bacnetModbusDamperInterop[1][22](
  AI_Volume					:= A_360_01_SQ5_C411_VOL,
  AV_CurrentSetpoint			:= A_360_01_SQ5_C411_SP,
  AV_vMin					:= A_360_01_SQ5_C411_VMIN,
  AV_vMax					:= A_360_01_SQ5_C411_VMAX,
  AI_Position				:= A_360_01_SQ5_C411_FB,
  AV_ControlledVariable		:= A_360_01_SQ5_C411_C,
  AV_ManualOverride			:= A_360_01_SQ5_C411_KMD,
  BV_ExcludeFromOptimizer	:= A_360_01_SQ5_C411_OPT_EKSKL,
  BV_DamperError				:= A_360_01_SQ5_C411_A1,
  BV_CommunicationError		:= A_360_01_SQ5_C411_A2,
  modbusHoldingRegisters		:= ADR(GVL_Modbus.awHoldingRegisters[i * 30]), 
  modbusCoilRegisters			:= ADR(GVL_Modbus.axCoils[i]), 
  typDamperInterface	    :=  GVL_Modbus.ModbusDamperInterface[1][22], 
  typDamperSettings       := PersistentVars.ModbusDamperSetpoints[1][22]
);
i := i +1;
// Kommunikasjonsalarmer

                
// Mappinger for spjeld +A=360.01-SK5A421

bacnetModbusDamperInterop[2][1](
  AI_Volume					:= A_360_01_SK5_A421_VOL,
  AV_CurrentSetpoint			:= A_360_01_SK5_A421_SP,
  AV_vMin					:= A_360_01_SK5_A421_VMIN,
  AV_vMax					:= A_360_01_SK5_A421_VMAX,
  AI_Position				:= A_360_01_SK5_A421_FB,
  AV_ControlledVariable		:= A_360_01_SK5_A421_C,
  AV_ManualOverride			:= A_360_01_SK5_A421_KMD,
  BV_ExcludeFromOptimizer	:= A_360_01_SK5_A421_OPT_EKSKL,
  BV_DamperError				:= A_360_01_SK5_A421_A1,
  BV_CommunicationError		:= A_360_01_SK5_A421_A2,
  modbusHoldingRegisters		:= ADR(GVL_Modbus.awHoldingRegisters[i * 30]), 
  modbusCoilRegisters			:= ADR(GVL_Modbus.axCoils[i]), 
  typDamperInterface	    :=  GVL_Modbus.ModbusDamperInterface[2][1], 
  typDamperSettings       := PersistentVars.ModbusDamperSetpoints[2][1]
);
i := i +1;
// Kommunikasjonsalarmer

                
// Mappinger for spjeld +A=360.01-SQ54AH2

bacnetModbusDamperInterop[2][2](
  AI_Volume					:= A_360_01_SQ5_4AH2_VOL,
  AV_CurrentSetpoint			:= A_360_01_SQ5_4AH2_SP,
  AV_vMin					:= A_360_01_SQ5_4AH2_VMIN,
  AV_vMax					:= A_360_01_SQ5_4AH2_VMAX,
  AI_Position				:= A_360_01_SQ5_4AH2_FB,
  AV_ControlledVariable		:= A_360_01_SQ5_4AH2_C,
  AV_ManualOverride			:= A_360_01_SQ5_4AH2_KMD,
  BV_ExcludeFromOptimizer	:= A_360_01_SQ5_4AH2_OPT_EKSKL,
  BV_DamperError				:= A_360_01_SQ5_4AH2_A1,
  BV_CommunicationError		:= A_360_01_SQ5_4AH2_A2,
  modbusHoldingRegisters		:= ADR(GVL_Modbus.awHoldingRegisters[i * 30]), 
  modbusCoilRegisters			:= ADR(GVL_Modbus.axCoils[i]), 
  typDamperInterface	    :=  GVL_Modbus.ModbusDamperInterface[2][2], 
  typDamperSettings       := PersistentVars.ModbusDamperSetpoints[2][2]
);
i := i +1;
// Kommunikasjonsalarmer

                
// Mappinger for spjeld +A=360.01-SK5A424

bacnetModbusDamperInterop[2][3](
  AI_Volume					:= A_360_01_SK5_A424_VOL,
  AV_CurrentSetpoint			:= A_360_01_SK5_A424_SP,
  AV_vMin					:= A_360_01_SK5_A424_VMIN,
  AV_vMax					:= A_360_01_SK5_A424_VMAX,
  AI_Position				:= A_360_01_SK5_A424_FB,
  AV_ControlledVariable		:= A_360_01_SK5_A424_C,
  AV_ManualOverride			:= A_360_01_SK5_A424_KMD,
  BV_ExcludeFromOptimizer	:= A_360_01_SK5_A424_OPT_EKSKL,
  BV_DamperError				:= A_360_01_SK5_A424_A1,
  BV_CommunicationError		:= A_360_01_SK5_A424_A2,
  modbusHoldingRegisters		:= ADR(GVL_Modbus.awHoldingRegisters[i * 30]), 
  modbusCoilRegisters			:= ADR(GVL_Modbus.axCoils[i]), 
  typDamperInterface	    :=  GVL_Modbus.ModbusDamperInterface[2][3], 
  typDamperSettings       := PersistentVars.ModbusDamperSetpoints[2][3]
);
i := i +1;
// Kommunikasjonsalarmer

                
// Mappinger for spjeld +A=360.01-SQ44AH3

bacnetModbusDamperInterop[2][4](
  AI_Volume					:= A_360_01_SQ4_4AH3_VOL,
  AV_CurrentSetpoint			:= A_360_01_SQ4_4AH3_SP,
  AV_vMin					:= A_360_01_SQ4_4AH3_VMIN,
  AV_vMax					:= A_360_01_SQ4_4AH3_VMAX,
  AI_Position				:= A_360_01_SQ4_4AH3_FB,
  AV_ControlledVariable		:= A_360_01_SQ4_4AH3_C,
  AV_ManualOverride			:= A_360_01_SQ4_4AH3_KMD,
  BV_ExcludeFromOptimizer	:= A_360_01_SQ4_4AH3_OPT_EKSKL,
  BV_DamperError				:= A_360_01_SQ4_4AH3_A1,
  BV_CommunicationError		:= A_360_01_SQ4_4AH3_A2,
  modbusHoldingRegisters		:= ADR(GVL_Modbus.awHoldingRegisters[i * 30]), 
  modbusCoilRegisters			:= ADR(GVL_Modbus.axCoils[i]), 
  typDamperInterface	    :=  GVL_Modbus.ModbusDamperInterface[2][4], 
  typDamperSettings       := PersistentVars.ModbusDamperSetpoints[2][4]
);
i := i +1;
// Kommunikasjonsalarmer

                
// Mappinger for spjeld +A=360.01-SQ44AH4

bacnetModbusDamperInterop[2][5](
  AI_Volume					:= A_360_01_SQ4_4AH4_VOL,
  AV_CurrentSetpoint			:= A_360_01_SQ4_4AH4_SP,
  AV_vMin					:= A_360_01_SQ4_4AH4_VMIN,
  AV_vMax					:= A_360_01_SQ4_4AH4_VMAX,
  AI_Position				:= A_360_01_SQ4_4AH4_FB,
  AV_ControlledVariable		:= A_360_01_SQ4_4AH4_C,
  AV_ManualOverride			:= A_360_01_SQ4_4AH4_KMD,
  BV_ExcludeFromOptimizer	:= A_360_01_SQ4_4AH4_OPT_EKSKL,
  BV_DamperError				:= A_360_01_SQ4_4AH4_A1,
  BV_CommunicationError		:= A_360_01_SQ4_4AH4_A2,
  modbusHoldingRegisters		:= ADR(GVL_Modbus.awHoldingRegisters[i * 30]), 
  modbusCoilRegisters			:= ADR(GVL_Modbus.axCoils[i]), 
  typDamperInterface	    :=  GVL_Modbus.ModbusDamperInterface[2][5], 
  typDamperSettings       := PersistentVars.ModbusDamperSetpoints[2][5]
);
i := i +1;
// Kommunikasjonsalarmer

                
// Mappinger for spjeld +A=360.01-SQ44AH5

bacnetModbusDamperInterop[2][6](
  AI_Volume					:= A_360_01_SQ4_4AH5_VOL,
  AV_CurrentSetpoint			:= A_360_01_SQ4_4AH5_SP,
  AV_vMin					:= A_360_01_SQ4_4AH5_VMIN,
  AV_vMax					:= A_360_01_SQ4_4AH5_VMAX,
  AI_Position				:= A_360_01_SQ4_4AH5_FB,
  AV_ControlledVariable		:= A_360_01_SQ4_4AH5_C,
  AV_ManualOverride			:= A_360_01_SQ4_4AH5_KMD,
  BV_ExcludeFromOptimizer	:= A_360_01_SQ4_4AH5_OPT_EKSKL,
  BV_DamperError				:= A_360_01_SQ4_4AH5_A1,
  BV_CommunicationError		:= A_360_01_SQ4_4AH5_A2,
  modbusHoldingRegisters		:= ADR(GVL_Modbus.awHoldingRegisters[i * 30]), 
  modbusCoilRegisters			:= ADR(GVL_Modbus.axCoils[i]), 
  typDamperInterface	    :=  GVL_Modbus.ModbusDamperInterface[2][6], 
  typDamperSettings       := PersistentVars.ModbusDamperSetpoints[2][6]
);
i := i +1;
// Kommunikasjonsalarmer

                
// Mappinger for spjeld +A=360.01-SQ54AH3

bacnetModbusDamperInterop[2][7](
  AI_Volume					:= A_360_01_SQ5_4AH3_VOL,
  AV_CurrentSetpoint			:= A_360_01_SQ5_4AH3_SP,
  AV_vMin					:= A_360_01_SQ5_4AH3_VMIN,
  AV_vMax					:= A_360_01_SQ5_4AH3_VMAX,
  AI_Position				:= A_360_01_SQ5_4AH3_FB,
  AV_ControlledVariable		:= A_360_01_SQ5_4AH3_C,
  AV_ManualOverride			:= A_360_01_SQ5_4AH3_KMD,
  BV_ExcludeFromOptimizer	:= A_360_01_SQ5_4AH3_OPT_EKSKL,
  BV_DamperError				:= A_360_01_SQ5_4AH3_A1,
  BV_CommunicationError		:= A_360_01_SQ5_4AH3_A2,
  modbusHoldingRegisters		:= ADR(GVL_Modbus.awHoldingRegisters[i * 30]), 
  modbusCoilRegisters			:= ADR(GVL_Modbus.axCoils[i]), 
  typDamperInterface	    :=  GVL_Modbus.ModbusDamperInterface[2][7], 
  typDamperSettings       := PersistentVars.ModbusDamperSetpoints[2][7]
);
i := i +1;
// Kommunikasjonsalarmer

                
// Mappinger for spjeld +A=360.01-SQ5A401

bacnetModbusDamperInterop[2][8](
  AI_Volume					:= A_360_01_SQ5_A401_VOL,
  AV_CurrentSetpoint			:= A_360_01_SQ5_A401_SP,
  AV_vMin					:= A_360_01_SQ5_A401_VMIN,
  AV_vMax					:= A_360_01_SQ5_A401_VMAX,
  AI_Position				:= A_360_01_SQ5_A401_FB,
  AV_ControlledVariable		:= A_360_01_SQ5_A401_C,
  AV_ManualOverride			:= A_360_01_SQ5_A401_KMD,
  BV_ExcludeFromOptimizer	:= A_360_01_SQ5_A401_OPT_EKSKL,
  BV_DamperError				:= A_360_01_SQ5_A401_A1,
  BV_CommunicationError		:= A_360_01_SQ5_A401_A2,
  modbusHoldingRegisters		:= ADR(GVL_Modbus.awHoldingRegisters[i * 30]), 
  modbusCoilRegisters			:= ADR(GVL_Modbus.axCoils[i]), 
  typDamperInterface	    :=  GVL_Modbus.ModbusDamperInterface[2][8], 
  typDamperSettings       := PersistentVars.ModbusDamperSetpoints[2][8]
);
i := i +1;
// Kommunikasjonsalarmer

                
// Mappinger for spjeld +A=360.01-SQ4A403

bacnetModbusDamperInterop[2][9](
  AI_Volume					:= A_360_01_SQ4_A403_VOL,
  AV_CurrentSetpoint			:= A_360_01_SQ4_A403_SP,
  AV_vMin					:= A_360_01_SQ4_A403_VMIN,
  AV_vMax					:= A_360_01_SQ4_A403_VMAX,
  AI_Position				:= A_360_01_SQ4_A403_FB,
  AV_ControlledVariable		:= A_360_01_SQ4_A403_C,
  AV_ManualOverride			:= A_360_01_SQ4_A403_KMD,
  BV_ExcludeFromOptimizer	:= A_360_01_SQ4_A403_OPT_EKSKL,
  BV_DamperError				:= A_360_01_SQ4_A403_A1,
  BV_CommunicationError		:= A_360_01_SQ4_A403_A2,
  modbusHoldingRegisters		:= ADR(GVL_Modbus.awHoldingRegisters[i * 30]), 
  modbusCoilRegisters			:= ADR(GVL_Modbus.axCoils[i]), 
  typDamperInterface	    :=  GVL_Modbus.ModbusDamperInterface[2][9], 
  typDamperSettings       := PersistentVars.ModbusDamperSetpoints[2][9]
);
i := i +1;
// Kommunikasjonsalarmer

                
// Mappinger for spjeld +A=360.01-SQ4A401_3

bacnetModbusDamperInterop[2][10](
  AI_Volume					:= A_360_01_SQ4_A401_3_VOL,
  AV_CurrentSetpoint			:= A_360_01_SQ4_A401_3_SP,
  AV_vMin					:= A_360_01_SQ4_A401_3_VMIN,
  AV_vMax					:= A_360_01_SQ4_A401_3_VMAX,
  AI_Position				:= A_360_01_SQ4_A401_3_FB,
  AV_ControlledVariable		:= A_360_01_SQ4_A401_3_C,
  AV_ManualOverride			:= A_360_01_SQ4_A401_3_KMD,
  BV_ExcludeFromOptimizer	:= A_360_01_SQ4_A401_3_OPT_EKSKL,
  BV_DamperError				:= A_360_01_SQ4_A401_3_A1,
  BV_CommunicationError		:= A_360_01_SQ4_A401_3_A2,
  modbusHoldingRegisters		:= ADR(GVL_Modbus.awHoldingRegisters[i * 30]), 
  modbusCoilRegisters			:= ADR(GVL_Modbus.axCoils[i]), 
  typDamperInterface	    :=  GVL_Modbus.ModbusDamperInterface[2][10], 
  typDamperSettings       := PersistentVars.ModbusDamperSetpoints[2][10]
);
i := i +1;
// Kommunikasjonsalarmer

                
// Mappinger for spjeld +A=360.01-SQ4A401_4

bacnetModbusDamperInterop[2][11](
  AI_Volume					:= A_360_01_SQ4_A401_4_VOL,
  AV_CurrentSetpoint			:= A_360_01_SQ4_A401_4_SP,
  AV_vMin					:= A_360_01_SQ4_A401_4_VMIN,
  AV_vMax					:= A_360_01_SQ4_A401_4_VMAX,
  AI_Position				:= A_360_01_SQ4_A401_4_FB,
  AV_ControlledVariable		:= A_360_01_SQ4_A401_4_C,
  AV_ManualOverride			:= A_360_01_SQ4_A401_4_KMD,
  BV_ExcludeFromOptimizer	:= A_360_01_SQ4_A401_4_OPT_EKSKL,
  BV_DamperError				:= A_360_01_SQ4_A401_4_A1,
  BV_CommunicationError		:= A_360_01_SQ4_A401_4_A2,
  modbusHoldingRegisters		:= ADR(GVL_Modbus.awHoldingRegisters[i * 30]), 
  modbusCoilRegisters			:= ADR(GVL_Modbus.axCoils[i]), 
  typDamperInterface	    :=  GVL_Modbus.ModbusDamperInterface[2][11], 
  typDamperSettings       := PersistentVars.ModbusDamperSetpoints[2][11]
);
i := i +1;
// Kommunikasjonsalarmer

                
// Mappinger for spjeld +A=360.01-SQ4A401_5

bacnetModbusDamperInterop[2][12](
  AI_Volume					:= A_360_01_SQ4_A401_5_VOL,
  AV_CurrentSetpoint			:= A_360_01_SQ4_A401_5_SP,
  AV_vMin					:= A_360_01_SQ4_A401_5_VMIN,
  AV_vMax					:= A_360_01_SQ4_A401_5_VMAX,
  AI_Position				:= A_360_01_SQ4_A401_5_FB,
  AV_ControlledVariable		:= A_360_01_SQ4_A401_5_C,
  AV_ManualOverride			:= A_360_01_SQ4_A401_5_KMD,
  BV_ExcludeFromOptimizer	:= A_360_01_SQ4_A401_5_OPT_EKSKL,
  BV_DamperError				:= A_360_01_SQ4_A401_5_A1,
  BV_CommunicationError		:= A_360_01_SQ4_A401_5_A2,
  modbusHoldingRegisters		:= ADR(GVL_Modbus.awHoldingRegisters[i * 30]), 
  modbusCoilRegisters			:= ADR(GVL_Modbus.axCoils[i]), 
  typDamperInterface	    :=  GVL_Modbus.ModbusDamperInterface[2][12], 
  typDamperSettings       := PersistentVars.ModbusDamperSetpoints[2][12]
);
i := i +1;
// Kommunikasjonsalarmer

                
// Mappinger for spjeld +A=360.01-SQ4A401_6

bacnetModbusDamperInterop[2][13](
  AI_Volume					:= A_360_01_SQ4_A401_6_VOL,
  AV_CurrentSetpoint			:= A_360_01_SQ4_A401_6_SP,
  AV_vMin					:= A_360_01_SQ4_A401_6_VMIN,
  AV_vMax					:= A_360_01_SQ4_A401_6_VMAX,
  AI_Position				:= A_360_01_SQ4_A401_6_FB,
  AV_ControlledVariable		:= A_360_01_SQ4_A401_6_C,
  AV_ManualOverride			:= A_360_01_SQ4_A401_6_KMD,
  BV_ExcludeFromOptimizer	:= A_360_01_SQ4_A401_6_OPT_EKSKL,
  BV_DamperError				:= A_360_01_SQ4_A401_6_A1,
  BV_CommunicationError		:= A_360_01_SQ4_A401_6_A2,
  modbusHoldingRegisters		:= ADR(GVL_Modbus.awHoldingRegisters[i * 30]), 
  modbusCoilRegisters			:= ADR(GVL_Modbus.axCoils[i]), 
  typDamperInterface	    :=  GVL_Modbus.ModbusDamperInterface[2][13], 
  typDamperSettings       := PersistentVars.ModbusDamperSetpoints[2][13]
);
i := i +1;
// Kommunikasjonsalarmer

                
// Mappinger for spjeld +A=360.01-SQ4A401_7

bacnetModbusDamperInterop[2][14](
  AI_Volume					:= A_360_01_SQ4_A401_7_VOL,
  AV_CurrentSetpoint			:= A_360_01_SQ4_A401_7_SP,
  AV_vMin					:= A_360_01_SQ4_A401_7_VMIN,
  AV_vMax					:= A_360_01_SQ4_A401_7_VMAX,
  AI_Position				:= A_360_01_SQ4_A401_7_FB,
  AV_ControlledVariable		:= A_360_01_SQ4_A401_7_C,
  AV_ManualOverride			:= A_360_01_SQ4_A401_7_KMD,
  BV_ExcludeFromOptimizer	:= A_360_01_SQ4_A401_7_OPT_EKSKL,
  BV_DamperError				:= A_360_01_SQ4_A401_7_A1,
  BV_CommunicationError		:= A_360_01_SQ4_A401_7_A2,
  modbusHoldingRegisters		:= ADR(GVL_Modbus.awHoldingRegisters[i * 30]), 
  modbusCoilRegisters			:= ADR(GVL_Modbus.axCoils[i]), 
  typDamperInterface	    :=  GVL_Modbus.ModbusDamperInterface[2][14], 
  typDamperSettings       := PersistentVars.ModbusDamperSetpoints[2][14]
);
i := i +1;
// Kommunikasjonsalarmer

                
// Mappinger for spjeld +A=360.01-SQ4A401_8

bacnetModbusDamperInterop[2][15](
  AI_Volume					:= A_360_01_SQ4_A401_8_VOL,
  AV_CurrentSetpoint			:= A_360_01_SQ4_A401_8_SP,
  AV_vMin					:= A_360_01_SQ4_A401_8_VMIN,
  AV_vMax					:= A_360_01_SQ4_A401_8_VMAX,
  AI_Position				:= A_360_01_SQ4_A401_8_FB,
  AV_ControlledVariable		:= A_360_01_SQ4_A401_8_C,
  AV_ManualOverride			:= A_360_01_SQ4_A401_8_KMD,
  BV_ExcludeFromOptimizer	:= A_360_01_SQ4_A401_8_OPT_EKSKL,
  BV_DamperError				:= A_360_01_SQ4_A401_8_A1,
  BV_CommunicationError		:= A_360_01_SQ4_A401_8_A2,
  modbusHoldingRegisters		:= ADR(GVL_Modbus.awHoldingRegisters[i * 30]), 
  modbusCoilRegisters			:= ADR(GVL_Modbus.axCoils[i]), 
  typDamperInterface	    :=  GVL_Modbus.ModbusDamperInterface[2][15], 
  typDamperSettings       := PersistentVars.ModbusDamperSetpoints[2][15]
);
i := i +1;
// Kommunikasjonsalarmer

                
// Mappinger for spjeld +A=360.01-SQ4A401_9

bacnetModbusDamperInterop[2][16](
  AI_Volume					:= A_360_01_SQ4_A401_9_VOL,
  AV_CurrentSetpoint			:= A_360_01_SQ4_A401_9_SP,
  AV_vMin					:= A_360_01_SQ4_A401_9_VMIN,
  AV_vMax					:= A_360_01_SQ4_A401_9_VMAX,
  AI_Position				:= A_360_01_SQ4_A401_9_FB,
  AV_ControlledVariable		:= A_360_01_SQ4_A401_9_C,
  AV_ManualOverride			:= A_360_01_SQ4_A401_9_KMD,
  BV_ExcludeFromOptimizer	:= A_360_01_SQ4_A401_9_OPT_EKSKL,
  BV_DamperError				:= A_360_01_SQ4_A401_9_A1,
  BV_CommunicationError		:= A_360_01_SQ4_A401_9_A2,
  modbusHoldingRegisters		:= ADR(GVL_Modbus.awHoldingRegisters[i * 30]), 
  modbusCoilRegisters			:= ADR(GVL_Modbus.axCoils[i]), 
  typDamperInterface	    :=  GVL_Modbus.ModbusDamperInterface[2][16], 
  typDamperSettings       := PersistentVars.ModbusDamperSetpoints[2][16]
);
i := i +1;
// Kommunikasjonsalarmer

                
// Mappinger for spjeld +A=360.01-SQ4A401_0

bacnetModbusDamperInterop[2][17](
  AI_Volume					:= A_360_01_SQ4_A401_0_VOL,
  AV_CurrentSetpoint			:= A_360_01_SQ4_A401_0_SP,
  AV_vMin					:= A_360_01_SQ4_A401_0_VMIN,
  AV_vMax					:= A_360_01_SQ4_A401_0_VMAX,
  AI_Position				:= A_360_01_SQ4_A401_0_FB,
  AV_ControlledVariable		:= A_360_01_SQ4_A401_0_C,
  AV_ManualOverride			:= A_360_01_SQ4_A401_0_KMD,
  BV_ExcludeFromOptimizer	:= A_360_01_SQ4_A401_0_OPT_EKSKL,
  BV_DamperError				:= A_360_01_SQ4_A401_0_A1,
  BV_CommunicationError		:= A_360_01_SQ4_A401_0_A2,
  modbusHoldingRegisters		:= ADR(GVL_Modbus.awHoldingRegisters[i * 30]), 
  modbusCoilRegisters			:= ADR(GVL_Modbus.axCoils[i]), 
  typDamperInterface	    :=  GVL_Modbus.ModbusDamperInterface[2][17], 
  typDamperSettings       := PersistentVars.ModbusDamperSetpoints[2][17]
);
i := i +1;
// Kommunikasjonsalarmer

                
// Mappinger for spjeld +A=360.01-SQ4A426

bacnetModbusDamperInterop[2][18](
  AI_Volume					:= A_360_01_SQ4_A426_VOL,
  AV_CurrentSetpoint			:= A_360_01_SQ4_A426_SP,
  AV_vMin					:= A_360_01_SQ4_A426_VMIN,
  AV_vMax					:= A_360_01_SQ4_A426_VMAX,
  AI_Position				:= A_360_01_SQ4_A426_FB,
  AV_ControlledVariable		:= A_360_01_SQ4_A426_C,
  AV_ManualOverride			:= A_360_01_SQ4_A426_KMD,
  BV_ExcludeFromOptimizer	:= A_360_01_SQ4_A426_OPT_EKSKL,
  BV_DamperError				:= A_360_01_SQ4_A426_A1,
  BV_CommunicationError		:= A_360_01_SQ4_A426_A2,
  modbusHoldingRegisters		:= ADR(GVL_Modbus.awHoldingRegisters[i * 30]), 
  modbusCoilRegisters			:= ADR(GVL_Modbus.axCoils[i]), 
  typDamperInterface	    :=  GVL_Modbus.ModbusDamperInterface[2][18], 
  typDamperSettings       := PersistentVars.ModbusDamperSetpoints[2][18]
);
i := i +1;
// Kommunikasjonsalarmer

                
// Mappinger for spjeld +A=360.01-SQ4A428_1

bacnetModbusDamperInterop[2][19](
  AI_Volume					:= A_360_01_SQ4_A428_1_VOL,
  AV_CurrentSetpoint			:= A_360_01_SQ4_A428_1_SP,
  AV_vMin					:= A_360_01_SQ4_A428_1_VMIN,
  AV_vMax					:= A_360_01_SQ4_A428_1_VMAX,
  AI_Position				:= A_360_01_SQ4_A428_1_FB,
  AV_ControlledVariable		:= A_360_01_SQ4_A428_1_C,
  AV_ManualOverride			:= A_360_01_SQ4_A428_1_KMD,
  BV_ExcludeFromOptimizer	:= A_360_01_SQ4_A428_1_OPT_EKSKL,
  BV_DamperError				:= A_360_01_SQ4_A428_1_A1,
  BV_CommunicationError		:= A_360_01_SQ4_A428_1_A2,
  modbusHoldingRegisters		:= ADR(GVL_Modbus.awHoldingRegisters[i * 30]), 
  modbusCoilRegisters			:= ADR(GVL_Modbus.axCoils[i]), 
  typDamperInterface	    :=  GVL_Modbus.ModbusDamperInterface[2][19], 
  typDamperSettings       := PersistentVars.ModbusDamperSetpoints[2][19]
);
i := i +1;
// Kommunikasjonsalarmer

                
// Mappinger for spjeld +A=360.01-SQ4A428_2

bacnetModbusDamperInterop[2][20](
  AI_Volume					:= A_360_01_SQ4_A428_2_VOL,
  AV_CurrentSetpoint			:= A_360_01_SQ4_A428_2_SP,
  AV_vMin					:= A_360_01_SQ4_A428_2_VMIN,
  AV_vMax					:= A_360_01_SQ4_A428_2_VMAX,
  AI_Position				:= A_360_01_SQ4_A428_2_FB,
  AV_ControlledVariable		:= A_360_01_SQ4_A428_2_C,
  AV_ManualOverride			:= A_360_01_SQ4_A428_2_KMD,
  BV_ExcludeFromOptimizer	:= A_360_01_SQ4_A428_2_OPT_EKSKL,
  BV_DamperError				:= A_360_01_SQ4_A428_2_A1,
  BV_CommunicationError		:= A_360_01_SQ4_A428_2_A2,
  modbusHoldingRegisters		:= ADR(GVL_Modbus.awHoldingRegisters[i * 30]), 
  modbusCoilRegisters			:= ADR(GVL_Modbus.axCoils[i]), 
  typDamperInterface	    :=  GVL_Modbus.ModbusDamperInterface[2][20], 
  typDamperSettings       := PersistentVars.ModbusDamperSetpoints[2][20]
);
i := i +1;
// Kommunikasjonsalarmer

                
// Mappinger for spjeld +A=360.01-SQ4A428_3

bacnetModbusDamperInterop[2][21](
  AI_Volume					:= A_360_01_SQ4_A428_3_VOL,
  AV_CurrentSetpoint			:= A_360_01_SQ4_A428_3_SP,
  AV_vMin					:= A_360_01_SQ4_A428_3_VMIN,
  AV_vMax					:= A_360_01_SQ4_A428_3_VMAX,
  AI_Position				:= A_360_01_SQ4_A428_3_FB,
  AV_ControlledVariable		:= A_360_01_SQ4_A428_3_C,
  AV_ManualOverride			:= A_360_01_SQ4_A428_3_KMD,
  BV_ExcludeFromOptimizer	:= A_360_01_SQ4_A428_3_OPT_EKSKL,
  BV_DamperError				:= A_360_01_SQ4_A428_3_A1,
  BV_CommunicationError		:= A_360_01_SQ4_A428_3_A2,
  modbusHoldingRegisters		:= ADR(GVL_Modbus.awHoldingRegisters[i * 30]), 
  modbusCoilRegisters			:= ADR(GVL_Modbus.axCoils[i]), 
  typDamperInterface	    :=  GVL_Modbus.ModbusDamperInterface[2][21], 
  typDamperSettings       := PersistentVars.ModbusDamperSetpoints[2][21]
);
i := i +1;
// Kommunikasjonsalarmer

                
// Mappinger for spjeld +A=360.01-SQ4A428_4

bacnetModbusDamperInterop[2][22](
  AI_Volume					:= A_360_01_SQ4_A428_4_VOL,
  AV_CurrentSetpoint			:= A_360_01_SQ4_A428_4_SP,
  AV_vMin					:= A_360_01_SQ4_A428_4_VMIN,
  AV_vMax					:= A_360_01_SQ4_A428_4_VMAX,
  AI_Position				:= A_360_01_SQ4_A428_4_FB,
  AV_ControlledVariable		:= A_360_01_SQ4_A428_4_C,
  AV_ManualOverride			:= A_360_01_SQ4_A428_4_KMD,
  BV_ExcludeFromOptimizer	:= A_360_01_SQ4_A428_4_OPT_EKSKL,
  BV_DamperError				:= A_360_01_SQ4_A428_4_A1,
  BV_CommunicationError		:= A_360_01_SQ4_A428_4_A2,
  modbusHoldingRegisters		:= ADR(GVL_Modbus.awHoldingRegisters[i * 30]), 
  modbusCoilRegisters			:= ADR(GVL_Modbus.axCoils[i]), 
  typDamperInterface	    :=  GVL_Modbus.ModbusDamperInterface[2][22], 
  typDamperSettings       := PersistentVars.ModbusDamperSetpoints[2][22]
);
i := i +1;
// Kommunikasjonsalarmer

                
// Mappinger for spjeld +A=360.01-SQ5A425

bacnetModbusDamperInterop[2][23](
  AI_Volume					:= A_360_01_SQ5_A425_VOL,
  AV_CurrentSetpoint			:= A_360_01_SQ5_A425_SP,
  AV_vMin					:= A_360_01_SQ5_A425_VMIN,
  AV_vMax					:= A_360_01_SQ5_A425_VMAX,
  AI_Position				:= A_360_01_SQ5_A425_FB,
  AV_ControlledVariable		:= A_360_01_SQ5_A425_C,
  AV_ManualOverride			:= A_360_01_SQ5_A425_KMD,
  BV_ExcludeFromOptimizer	:= A_360_01_SQ5_A425_OPT_EKSKL,
  BV_DamperError				:= A_360_01_SQ5_A425_A1,
  BV_CommunicationError		:= A_360_01_SQ5_A425_A2,
  modbusHoldingRegisters		:= ADR(GVL_Modbus.awHoldingRegisters[i * 30]), 
  modbusCoilRegisters			:= ADR(GVL_Modbus.axCoils[i]), 
  typDamperInterface	    :=  GVL_Modbus.ModbusDamperInterface[2][23], 
  typDamperSettings       := PersistentVars.ModbusDamperSetpoints[2][23]
);
i := i +1;
// Kommunikasjonsalarmer

                
// Mappinger for spjeld +A=360.01-SQ4A428_5

bacnetModbusDamperInterop[2][24](
  AI_Volume					:= A_360_01_SQ4_A428_5_VOL,
  AV_CurrentSetpoint			:= A_360_01_SQ4_A428_5_SP,
  AV_vMin					:= A_360_01_SQ4_A428_5_VMIN,
  AV_vMax					:= A_360_01_SQ4_A428_5_VMAX,
  AI_Position				:= A_360_01_SQ4_A428_5_FB,
  AV_ControlledVariable		:= A_360_01_SQ4_A428_5_C,
  AV_ManualOverride			:= A_360_01_SQ4_A428_5_KMD,
  BV_ExcludeFromOptimizer	:= A_360_01_SQ4_A428_5_OPT_EKSKL,
  BV_DamperError				:= A_360_01_SQ4_A428_5_A1,
  BV_CommunicationError		:= A_360_01_SQ4_A428_5_A2,
  modbusHoldingRegisters		:= ADR(GVL_Modbus.awHoldingRegisters[i * 30]), 
  modbusCoilRegisters			:= ADR(GVL_Modbus.axCoils[i]), 
  typDamperInterface	    :=  GVL_Modbus.ModbusDamperInterface[2][24], 
  typDamperSettings       := PersistentVars.ModbusDamperSetpoints[2][24]
);
i := i +1;
// Kommunikasjonsalarmer

                
// Mappinger for spjeld +A=360.01-SQ4A428_6

bacnetModbusDamperInterop[2][25](
  AI_Volume					:= A_360_01_SQ4_A428_6_VOL,
  AV_CurrentSetpoint			:= A_360_01_SQ4_A428_6_SP,
  AV_vMin					:= A_360_01_SQ4_A428_6_VMIN,
  AV_vMax					:= A_360_01_SQ4_A428_6_VMAX,
  AI_Position				:= A_360_01_SQ4_A428_6_FB,
  AV_ControlledVariable		:= A_360_01_SQ4_A428_6_C,
  AV_ManualOverride			:= A_360_01_SQ4_A428_6_KMD,
  BV_ExcludeFromOptimizer	:= A_360_01_SQ4_A428_6_OPT_EKSKL,
  BV_DamperError				:= A_360_01_SQ4_A428_6_A1,
  BV_CommunicationError		:= A_360_01_SQ4_A428_6_A2,
  modbusHoldingRegisters		:= ADR(GVL_Modbus.awHoldingRegisters[i * 30]), 
  modbusCoilRegisters			:= ADR(GVL_Modbus.axCoils[i]), 
  typDamperInterface	    :=  GVL_Modbus.ModbusDamperInterface[2][25], 
  typDamperSettings       := PersistentVars.ModbusDamperSetpoints[2][25]
);
i := i +1;
// Kommunikasjonsalarmer

                
// Mappinger for spjeld +A=360.01-SQ4A428_7

bacnetModbusDamperInterop[2][26](
  AI_Volume					:= A_360_01_SQ4_A428_7_VOL,
  AV_CurrentSetpoint			:= A_360_01_SQ4_A428_7_SP,
  AV_vMin					:= A_360_01_SQ4_A428_7_VMIN,
  AV_vMax					:= A_360_01_SQ4_A428_7_VMAX,
  AI_Position				:= A_360_01_SQ4_A428_7_FB,
  AV_ControlledVariable		:= A_360_01_SQ4_A428_7_C,
  AV_ManualOverride			:= A_360_01_SQ4_A428_7_KMD,
  BV_ExcludeFromOptimizer	:= A_360_01_SQ4_A428_7_OPT_EKSKL,
  BV_DamperError				:= A_360_01_SQ4_A428_7_A1,
  BV_CommunicationError		:= A_360_01_SQ4_A428_7_A2,
  modbusHoldingRegisters		:= ADR(GVL_Modbus.awHoldingRegisters[i * 30]), 
  modbusCoilRegisters			:= ADR(GVL_Modbus.axCoils[i]), 
  typDamperInterface	    :=  GVL_Modbus.ModbusDamperInterface[2][26], 
  typDamperSettings       := PersistentVars.ModbusDamperSetpoints[2][26]
);
i := i +1;
// Kommunikasjonsalarmer

                
// Mappinger for spjeld +B=360.02-SQ5UBH1

bacnetModbusDamperInterop[3][1](
  AI_Volume					:= B_360_02_SQ5_UBH1_VOL,
  AV_CurrentSetpoint			:= B_360_02_SQ5_UBH1_SP,
  AV_vMin					:= B_360_02_SQ5_UBH1_VMIN,
  AV_vMax					:= B_360_02_SQ5_UBH1_VMAX,
  AI_Position				:= B_360_02_SQ5_UBH1_FB,
  AV_ControlledVariable		:= B_360_02_SQ5_UBH1_C,
  AV_ManualOverride			:= B_360_02_SQ5_UBH1_KMD,
  BV_ExcludeFromOptimizer	:= B_360_02_SQ5_UBH1_OPT_EKSKL,
  BV_DamperError				:= B_360_02_SQ5_UBH1_A1,
  BV_CommunicationError		:= B_360_02_SQ5_UBH1_A2,
  modbusHoldingRegisters		:= ADR(GVL_Modbus.awHoldingRegisters[i * 30]), 
  modbusCoilRegisters			:= ADR(GVL_Modbus.axCoils[i]), 
  typDamperInterface	    :=  GVL_Modbus.ModbusDamperInterface[3][1], 
  typDamperSettings       := PersistentVars.ModbusDamperSetpoints[3][1]
);
i := i +1;
// Kommunikasjonsalarmer

                
// Mappinger for spjeld +B=360.02-SQ5UBH2

bacnetModbusDamperInterop[3][2](
  AI_Volume					:= B_360_02_SQ5_UBH2_VOL,
  AV_CurrentSetpoint			:= B_360_02_SQ5_UBH2_SP,
  AV_vMin					:= B_360_02_SQ5_UBH2_VMIN,
  AV_vMax					:= B_360_02_SQ5_UBH2_VMAX,
  AI_Position				:= B_360_02_SQ5_UBH2_FB,
  AV_ControlledVariable		:= B_360_02_SQ5_UBH2_C,
  AV_ManualOverride			:= B_360_02_SQ5_UBH2_KMD,
  BV_ExcludeFromOptimizer	:= B_360_02_SQ5_UBH2_OPT_EKSKL,
  BV_DamperError				:= B_360_02_SQ5_UBH2_A1,
  BV_CommunicationError		:= B_360_02_SQ5_UBH2_A2,
  modbusHoldingRegisters		:= ADR(GVL_Modbus.awHoldingRegisters[i * 30]), 
  modbusCoilRegisters			:= ADR(GVL_Modbus.axCoils[i]), 
  typDamperInterface	    :=  GVL_Modbus.ModbusDamperInterface[3][2], 
  typDamperSettings       := PersistentVars.ModbusDamperSetpoints[3][2]
);
i := i +1;
// Kommunikasjonsalarmer

                
// Mappinger for spjeld +B=360.02-SQ4UBH1

bacnetModbusDamperInterop[3][3](
  AI_Volume					:= B_360_02_SQ4_UBH1_VOL,
  AV_CurrentSetpoint			:= B_360_02_SQ4_UBH1_SP,
  AV_vMin					:= B_360_02_SQ4_UBH1_VMIN,
  AV_vMax					:= B_360_02_SQ4_UBH1_VMAX,
  AI_Position				:= B_360_02_SQ4_UBH1_FB,
  AV_ControlledVariable		:= B_360_02_SQ4_UBH1_C,
  AV_ManualOverride			:= B_360_02_SQ4_UBH1_KMD,
  BV_ExcludeFromOptimizer	:= B_360_02_SQ4_UBH1_OPT_EKSKL,
  BV_DamperError				:= B_360_02_SQ4_UBH1_A1,
  BV_CommunicationError		:= B_360_02_SQ4_UBH1_A2,
  modbusHoldingRegisters		:= ADR(GVL_Modbus.awHoldingRegisters[i * 30]), 
  modbusCoilRegisters			:= ADR(GVL_Modbus.axCoils[i]), 
  typDamperInterface	    :=  GVL_Modbus.ModbusDamperInterface[3][3], 
  typDamperSettings       := PersistentVars.ModbusDamperSetpoints[3][3]
);
i := i +1;
// Kommunikasjonsalarmer

                
// Mappinger for spjeld +B=360.02-SQ4UBH2

bacnetModbusDamperInterop[3][4](
  AI_Volume					:= B_360_02_SQ4_UBH2_VOL,
  AV_CurrentSetpoint			:= B_360_02_SQ4_UBH2_SP,
  AV_vMin					:= B_360_02_SQ4_UBH2_VMIN,
  AV_vMax					:= B_360_02_SQ4_UBH2_VMAX,
  AI_Position				:= B_360_02_SQ4_UBH2_FB,
  AV_ControlledVariable		:= B_360_02_SQ4_UBH2_C,
  AV_ManualOverride			:= B_360_02_SQ4_UBH2_KMD,
  BV_ExcludeFromOptimizer	:= B_360_02_SQ4_UBH2_OPT_EKSKL,
  BV_DamperError				:= B_360_02_SQ4_UBH2_A1,
  BV_CommunicationError		:= B_360_02_SQ4_UBH2_A2,
  modbusHoldingRegisters		:= ADR(GVL_Modbus.awHoldingRegisters[i * 30]), 
  modbusCoilRegisters			:= ADR(GVL_Modbus.axCoils[i]), 
  typDamperInterface	    :=  GVL_Modbus.ModbusDamperInterface[3][4], 
  typDamperSettings       := PersistentVars.ModbusDamperSetpoints[3][4]
);
i := i +1;
// Kommunikasjonsalarmer

                
              
END_PROGRAM
